ABB RAPID module: MainModule.mod

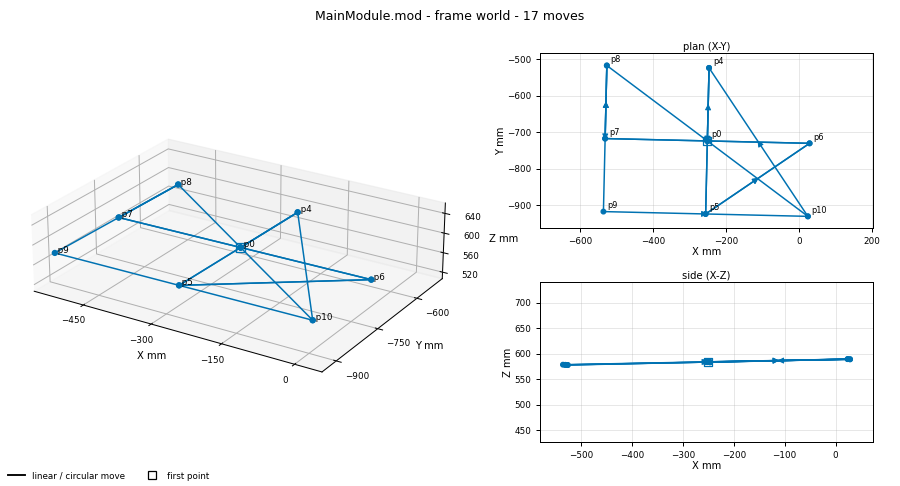
[picture p0: tool path of MainModule.mod in frame world, 17 of 17 moves have a stored position in this frame; points joined in program order, loops and branches not executed]
MODULE MainModule
	LOCAL CONST robtarget p0:=[[-251.2,-723.77,583.73],[0.00762991,0.715272,0.698776,0.00625841],[-2,-4,-1,0],[9E+09,9E+09,9E+09,9E+09,9E+09,9E+09]];
	LOCAL CONST robtarget p1:=[[-251.2,-723.77,583.73],[0.00982053,0.0116644,0.999883,-0.000969797],[-2,-4,-1,0],[9E+09,9E+09,9E+09,9E+09,9E+09,9E+09]];
	LOCAL CONST robtarget p2:=[[-251.2,-723.77,583.73],[0.000969797,0.999883,-0.0116644,0.00982053],[-2,-4,-1,0],[9E+09,9E+09,9E+09,9E+09,9E+09,9E+09]];
	LOCAL CONST robtarget p3:=[[-251.2,-723.77,583.73],[0.00625841,-0.698776,0.715272,-0.00762991],[-2,-4,-1,0],[9E+09,9E+09,9E+09,9E+09,9E+09,9E+09]];
	LOCAL CONST robtarget p4:=[[-246.535,-524.003,583.388],[0.188227,0.69252,0.672991,-0.179081],[-2,-4,-1,0],[9E+09,9E+09,9E+09,9E+09,9E+09,9E+09]];
	LOCAL CONST robtarget p5:=[[-255.865,-923.537,584.072],[-0.173487,0.68928,0.676941,0.191171],[-2,-4,-1,0],[9E+09,9E+09,9E+09,9E+09,9E+09,9E+09]];
	LOCAL CONST robtarget p6:=[[28.4199,-730.29,589.23],[-0.177756,0.692875,0.676586,-0.174811],[-2,-4,-1,0],[9E+09,9E+09,9E+09,9E+09,9E+09,9E+09]];
	LOCAL CONST robtarget p7:=[[-530.82,-717.25,578.23],[0.192496,0.688925,0.673346,0.186902],[-2,-4,-1,0],[9E+09,9E+09,9E+09,9E+09,9E+09,9E+09]];
	LOCAL CONST robtarget p8:=[[-526.155,-517.483,577.888],[0.36105,0.620206,0.696409,0.00120407],[-2,-4,-1,0],[9E+09,9E+09,9E+09,9E+09,9E+09,9E+09]];
	LOCAL CONST robtarget p9:=[[-535.485,-917.017,578.571],[0.0108236,0.710695,0.604396,0.359862],[-2,-4,-1,0],[9E+09,9E+09,9E+09,9E+09,9E+09,9E+09]];
	LOCAL CONST robtarget p10:=[[23.755,-930.057,589.572],[-0.345974,0.620892,0.703353,0.00945207],[-2,-4,-1,0],[9E+09,9E+09,9E+09,9E+09,9E+09,9E+09]];
	LOCAL CONST robtarget p11:=[[33.0848,-530.523,588.889],[0.00257557,0.717639,0.60371,-0.347162],[-2,-4,-1,0],[9E+09,9E+09,9E+09,9E+09,9E+09,9E+09]];
	LOCAL CONST robtarget p12:=[[-246.535,-524.003,583.388],[0.259726,0.965562,-0.0138087,0.00646692],[-2,-4,-1,0],[9E+09,9E+09,9E+09,9E+09,9E+09,9E+09]];
	LOCAL CONST robtarget p13:=[[-255.865,-923.537,584.072],[-0.257852,0.966064,-0.00872524,0.0125049],[-2,-4,-1,0],[9E+09,9E+09,9E+09,9E+09,9E+09,9E+09]];
	LOCAL CONST robtarget p14:=[[28.4199,-730.29,589.23],[-0.00208223,0.968355,-0.011518,-0.249303],[-2,-4,-1,0],[9E+09,9E+09,9E+09,9E+09,9E+09,9E+09]];
	LOCAL CONST robtarget p15:=[[-530.82,-717.25,578.23],[0.00395573,0.963271,-0.011016,0.268275],[-2,-4,-1,0],[9E+09,9E+09,9E+09,9E+09,9E+09,9E+09]];
	LOCAL CONST robtarget p16:=[[-526.155,-517.483,577.888],[0.25445,0.930988,0.0538837,0.256152],[-2,-4,-1,0],[9E+09,9E+09,9E+09,9E+09,9E+09,9E+09]];
	LOCAL CONST robtarget p17:=[[-535.485,-917.017,578.571],[-0.246808,0.92991,-0.0751649,0.262115],[-2,-4,-1,0],[9E+09,9E+09,9E+09,9E+09,9E+09,9E+09]];
	LOCAL CONST robtarget p18:=[[23.755,-930.057,589.572],[-0.251324,0.936383,0.0583091,-0.237957],[-2,-4,-1,0],[9E+09,9E+09,9E+09,9E+09,9E+09,9E+09]];
	LOCAL CONST robtarget p19:=[[33.0848,-530.523,588.889],[0.247302,0.934335,-0.0805601,-0.243659],[-2,-4,-1,0],[9E+09,9E+09,9E+09,9E+09,9E+09,9E+09]];

	LOCAL CONST wobjdata wobj_charuco:=[FALSE,TRUE,"",[[82.8438,-884.479,38.2097],[0.706341,-0.00783969,-0.00137015,0.707827]],[[0,0,0],[1,0,0,0]]];

	LOCAL CONST tooldata camera:=[TRUE,[[-16.651746849288683, 237.13801801978257, 158.9293391764847],[0.7121831587768082, -0.0053121823096013866, -0.7018028633858873, -0.01548127957138288 ]],[-1,[0,0,0],[1,0,0,0],0,0,0]];

	PROC main()
		MoveL p0, v100, z50, tool0;
		MoveL p1, v100, z50, tool0;
		MoveL p2, v100, z50, tool0;
		MoveL p3, v100, z50, tool0;
		MoveL p4, v100, z50, tool0;
		MoveL p5, v100, z50, tool0;
		MoveL p6, v100, z50, tool0;
		MoveL p7, v100, z50, tool0;
		MoveL p8, v100, z50, tool0;
		MoveL p9, v100, z50, tool0;
		MoveL p10, v100, z50, tool0;
		!MoveL p11, v100, z50, tool0;
		MoveL p12, v100, z50, tool0;
		MoveL p13, v100, z50, tool0;
		MoveL p14, v100, z50, tool0;
		MoveL p15, v100, z50, tool0;
		MoveL p16, v100, z50, tool0;
		!MoveL p17, v100, z50, tool0;
		MoveL p18, v100, z50, tool0;
		!MoveL p19, v100, z50, tool0;
	ENDPROC
ENDMODULE
